// TwinCAT 3 PLC project Analog_Voltage_Input
// ProgramVersion: 3.1.4023.0
// libraries:
//   Tc2_Standard, * (Beckhoff Automation GmbH)
//   Tc2_System, * (Beckhoff Automation GmbH)
//   Tc3_Module, * (Beckhoff Automation GmbH)
// project tree:
//   GVLs/ GVL.TcGVL
//   / PlcTask.TcTTO
//   POUs/ MAIN.TcPOU, ReadAnalogInput.TcPOU, ReadAnalogInputST.TcPOU
// real-time tasks:
//   TASK PlcTask: cycle T#10ms, priority 20, ADS port 350
// I/O:
//   DEVICE Dispositivo 1 (EtherCAT), AmsNetId 5.71.198.244.2.1
//     Terminale 1 (EK1200) [EK1200-5000 EtherCAT Power supply (2A E-Bus)]
//       Terminale 2 (EL2008) [EL2008 8Ch. Dig. Output 24V, 0.5A]
//       Terminale 3 (EL1008) [EL1008 8Ch. Dig. Input 24V, 3ms]
//       Terminale 4 (EL3064) [EL3064 4Ch. Ana. Input 0-10V]
//       Terminale 5 (EL9011) [EL9011 End Terminal]
// variable links:
//   Analog_Voltage_Input/Analog_Voltage_Input Instance <-> Device 1 (EtherCAT)/Term 1 (EK1200)/Term 4 (EL3064)
//     PlcTask Inputs/GVL.Analog_Inputs[1] <-> AI Standard Channel 1/Value

CONFIGURATION Analog_Voltage_Input
    RESOURCE PLC ON TwinCAT3
        TASK PlcTask(INTERVAL := T#10ms, PRIORITY := 20);
        PROGRAM MAIN WITH PlcTask : MAIN;
    END_RESOURCE
END_CONFIGURATION

// ---- GVLs/GVL.TcGVL
{attribute 'qualified_only'}
VAR_GLOBAL
	Analog_Inputs AT %I* : ARRAY[1..4] OF INT;
	Analog_Inputs_Values : ARRAY[1..4] OF REAL;
END_VAR

// ---- POUs/MAIN.TcPOU
PROGRAM MAIN
VAR
END_VAR

ReadAnalogInput();

END_PROGRAM

// ---- POUs/ReadAnalogInput.TcPOU
PROGRAM ReadAnalogInput
VAR
	Temp: REAL;
END_VAR

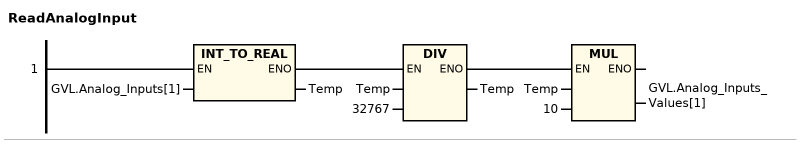
// NETWORK 1
Temp := INT_TO_REAL(GVL.Analog_Inputs[1]);
Temp := Temp / 32767;
GVL.Analog_Inputs_Values[1] := Temp * 10;

END_PROGRAM

// ---- POUs/ReadAnalogInputST.TcPOU
PROGRAM ReadAnalogInputST
VAR
END_VAR

GVL.Analog_Inputs_Values[1] := INT_TO_REAL(GVL.Analog_Inputs[1])/32767*10;
GVL.Analog_Inputs_Values[2] := INT_TO_REAL(GVL.Analog_Inputs[2])/32767*10;
GVL.Analog_Inputs_Values[3] := INT_TO_REAL(GVL.Analog_Inputs[3])/32767*10;
GVL.Analog_Inputs_Values[4] := INT_TO_REAL(GVL.Analog_Inputs[4])/32767*10;

END_PROGRAM
